// TwinCAT 3 PLC project Alarmbewaking
// ProgramVersion: 3.1.4024.0
// libraries:
//   Tc2_Standard, * (Beckhoff Automation GmbH)
//   Tc2_System, * (Beckhoff Automation GmbH)
//   Tc3_Module, * (Beckhoff Automation GmbH)
// project tree:
//   / PlcTask.TcTTO
//   POUs/ MAIN.TcPOU
// (motion and I/O tree: see PLC project potentiometer_inlezen)
// real-time tasks:
//   TASK PlcTask: cycle T#10ms, priority 20, ADS port 350
//   TASK PlcTask1: cycle T#10ms, priority 21, ADS port 351
//   TASK PlcTask2: cycle T#10ms, priority 22, ADS port 352
//   TASK PlcTask3: cycle T#10ms, priority 26, ADS port 353
//   TASK PlcTask4: cycle T#10ms, priority 25, ADS port 354
//   TASK PlcTask5: cycle T#10ms, priority 24, ADS port 355
//   TASK PlcTask6: cycle T#10ms, priority 23, ADS port 356
//   TASK PlcTask7: cycle T#10ms, priority 27, ADS port 357

CONFIGURATION Alarmbewaking
    RESOURCE PLC ON TwinCAT3
        TASK PlcTask(INTERVAL := T#10ms, PRIORITY := 26);
        PROGRAM MAIN WITH PlcTask : MAIN;
    END_RESOURCE
END_CONFIGURATION

// ---- POUs/MAIN.TcPOU
PROGRAM MAIN
VAR
	
// Inputs	
	druk: INT;
	temperatuur: INT;
	niveau: INT;
	
// Outputs	
	Lamp1: BOOL;
	Lamp2: BOOL;
	Lamp3: BOOL;
	Lamp4: BOOL;
	Lamp5: BOOL;
END_VAR

(*
Alarmbewaking (5 regels code)

We herhalen de oefening van de alarmbewaking. We maken nu echter gebruik van simpele analoge sensoren. 
We moeten nu de drempelwaarden die we normaal in onze smart sensor zouden ingesteld hebben aan het programma moeten meegeven. 
Deze zijn voor de druk, temperatuur en vloeistofniveau respectievelijk 12, 80 en 22. 
Het programma dat we geschreven hebben voor onze 5 lampen blijft zo goed als hetzelfde.
*)
Lamp1 := druk > 12;
Lamp2 := temperatuur > 80;
Lamp3 := niveau < 22;
Lamp4 := (Lamp1 AND Lamp2) OR (Lamp1 AND Lamp3) OR (Lamp2 AND Lamp3);
Lamp5 := Lamp1 AND Lamp2 AND Lamp3;

END_PROGRAM
